// TIA Portal V19 export
DATA_BLOCK "OP"   // DB29
{ S7_Optimized_Access := 'FALSE' }
   VAR
      HOOTER : Bool;
      "PUMP-1" : Bool;
      "PUMP-2" : Bool;
      DS_PUMP : Bool;
      "PNV-1" : Bool;
      "PNV-2" : Bool;
      "PNV-3" : Bool;
      "PNV-4" : Bool;
      "PNV-5" : Bool;
      "PNV-6" : Bool;
      "PNV-7" : Bool;
      "PNV-8" : Bool;
      "PNV-9" : Bool;
      "PNV-10" : Bool;
      "PNV-11" : Bool;
      "PNV-12" : Bool;
      "PNV-13" : Bool;
      "PNV-14" : Bool;
      "PNV-15" : Bool;
      "PNV-16" : Bool;
      "PNV-17" : Bool;
      "PNV-18" : Bool;
      "PNV-19" : Bool;
      "PNV-20" : Bool;
      "PNV-21" : Bool;
      "PNV-22" : Bool;
      "PZDV-1" : Bool;
      "PZDV-2" : Bool;
      CIP_IN : Bool;
      CIP_OUT : Bool;
      "PNV-25" : Bool;
   END_VAR
BEGIN
END_DATA_BLOCK
